DATA_BLOCK "ID_Algemeen_CM_DI_iDkReset"
{ S7_Optimized_Access := 'FALSE' }
VERSION : 0.1
NON_RETAIN
"FB_CM_DI_Sensor"

BEGIN

END_DATA_BLOCK

